PROGRAM IO
VAR
END_VAR

Term06();

Term07();

END_PROGRAM

(* stored: Version 1.1.0.1
   POU IO: Id {a0340162-3608-4e28-bda3-2d06c9afbd18}, SpecialFunc None *)
